{attribute 'GeneratedUsingTerminal: EL3783-0000-0018'}
{attribute addProperty BoxType "EL3783-0000-0018"}
{attribute addProperty Id "HCR_0USINT1HCR_1USINT1HCR_2USINT1HCR_3USINT1"}
{attribute addProperty CRC "1217820514"}
{attribute addProperty Size "4"}
TYPE High_Current_Range_48967762 :
STRUCT
	{attribute addProperty Name "HCR_0"}
	HCR_0 : USINT;
	{attribute addProperty Name "HCR_1"}
	HCR_1 : USINT;
	{attribute addProperty Name "HCR_2"}
	HCR_2 : USINT;
	{attribute addProperty Name "HCR_3"}
	HCR_3 : USINT;
END_STRUCT
END_TYPE

(* stored: Version 1.2.0.0, ProductVersion 3.1.4024.11
   DUT High_Current_Range_48967762: Id {ef8ae030-f7f6-4fe6-a580-e4d074c6f50f} *)
